TYPE csp_main_accuChange_enum :
(
	CSP_MAIN_ACCUCHANGE_STATUS_BRAND_CHECK 									:= 0,
	CSP_MAIN_ACCUCHANGE_STATUS_BRAND_CHANGE_REQUEST 						:= 5,
	CSP_MAIN_ACCUCHANGE_STATUS_PRODUCT_REMOVED_CHECK 						:= 10,
	CSP_MAIN_ACCUCHANGE_STATUS_RESET_REQUEST								:= 20,
	CSP_MAIN_ACCUCHANGE_STATUS_SAFE_POSITION_REQUEST 						:= 30,
	CSP_MAIN_ACCUCHANGE_STATUS_OPERATOR_REPLACE_CHANGE_PARTS 				:= 40,
	CSP_MAIN_ACCUCHANGE_STATUS_CHANGE_PARTS_REPLACED						:= 50,
	CSP_MAIN_ACCUCHANGE_STATUS_VERIFYING_CHANGE_PARTS_START					:= 60,
	CSP_MAIN_ACCUCHANGE_STATUS_VERIFYING_CASE_FEED_EOAT						:= 61,
	CSP_MAIN_ACCUCHANGE_STATUS_VERIFYING_LOADER_PUSHER						:= 62,
	CSP_MAIN_ACCUCHANGE_STATUS_VERIFYING_LOADER_GUIDE_PLATE					:= 63,
	CSP_MAIN_ACCUCHANGE_STATUS_VERIFYING_CLOSING_PADDLES					:= 64,
	CSP_MAIN_ACCUCHANGE_STATUS_VERIFYING_ALL_RFID							:= 65,
	CSP_MAIN_ACCUCHANGE_STATUS_GROUP_1_ACCU_MOVE_REQUEST 					:= 70,
	CSP_MAIN_ACCUCHANGE_STATUS_GROUP_2_TR_UP_ACCU_MOVE_REQUEST 				:= 80,
	CSP_MAIN_ACCUCHANGE_STATUS_GROUP_2_TR_DOWN_ACCU_MOVE_REQUEST 			:= 85,
	CSP_MAIN_ACCUCHANGE_STATUS_ADD_CASE_BLANKS 								:= 100,
	CSP_MAIN_ACCUCHANGE_STATUS_DONE											:= 900
) := CSP_MAIN_ACCUCHANGE_STATUS_BRAND_CHECK;
END_TYPE

(* stored: Version 1.1.0.1, ProductVersion 3.1.4024.3
   DUT csp_main_accuChange_enum: Id {498b916c-a397-4896-8e14-ecee1b070df8} *)
